PROGRAM p10_directionalInterlock
VAR
	interlockS0: TOF;
	interlockS1: TOF;
	S0: BOOL;	
	S1: BOOL;
	L0: BOOL;
	L1: BOOL;
END_VAR

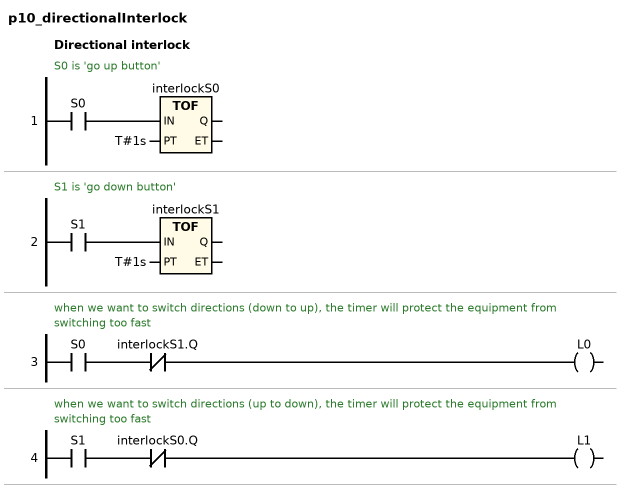
// NETWORK 1: Directional interlock
// S0 is 'go up button'
interlockS0(IN := S0, PT := T#1s); // TOF

// NETWORK 2
// S1 is 'go down button'
interlockS1(IN := S1, PT := T#1s); // TOF

// NETWORK 3
// when we want to switch directions (down to up), the timer will protect the equipment from switching too fast
L0 := S0 AND NOT interlockS1.Q;

// NETWORK 4
// when we want to switch directions (up to down), the timer will protect the equipment from switching too fast
L1 := S1 AND NOT interlockS0.Q;

END_PROGRAM

(* stored: Version 1.1.0.1, ProductVersion 3.1.4024.13
   POU p10_directionalInterlock: Id {b3c8980f-3d02-4274-af18-ef452a29b063}, SpecialFunc None *)
